PROGRAM Bottle_Filling_System
VAR
	Sensor: BOOL;
	Valve: BOOL;
	TOF_0: TOF;
END_VAR

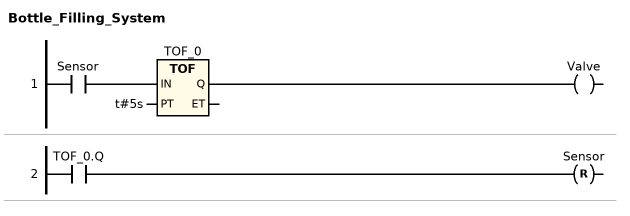
// NETWORK 1
TOF_0(IN := Sensor, PT := t#5s); // TOF
Valve := TOF_0.Q;

// NETWORK 2
Sensor R= TOF_0.Q;

END_PROGRAM

(* stored: Version 1.1.0.1, ProductVersion 3.1.4024.11
   POU Bottle_Filling_System: Id {ecb527ef-d2bb-4f15-885a-b22e200e3632}, SpecialFunc None *)
